// Brief: Master Arm Master Slave Control
FUNCTION_BLOCK PUBLIC FB_StateCtrlInit EXTENDS FB_MasterArmCtrlBase
VAR_INPUT
END_VAR
VAR_OUTPUT
END_VAR
VAR

END_VAR

// override this function in each exact controller
METHOD PROTECTED calcCmdJntPos : BOOL

VAR_IN_OUT CONSTANT
	i_slaveIdx :INT;
	i_shoulderPose :ST_Frame;
	i_masterArm :FB_MasterArm;
	i_slaveStatus :ST_SlaveStatus;
END_VAR

VAR
	centerVel:LREAL;
//	curJntPos:Vec7d;
END_VAR
IF m_isFinished THEN
	RETURN;
END_IF

IF m_timePeriod > 1 THEN
	m_isFinished :=true;
END_IF
END_METHOD

METHOD PUBLIC init : BOOL
VAR_IN_OUT CONSTANT
	i_masterArm	:FB_MasterArm;
END_VAR
VAR_IN_OUT 
	r_masterArmCtrlCmd :ST_ArmCtrlCmds;
END_VAR

VAR
	i:INT;
END_VAR
SUPER^.Init(i_masterArm,r_masterArmCtrlCmd);
m_jntEnableFlag :=g_zeroVec7i;
END_METHOD

END_FUNCTION_BLOCK

(* stored: Version 1.1.0.1, ProductVersion 3.1.4024.11
   POU FB_StateCtrlInit: Id {2f1b91d8-ebd5-4b63-92d8-450fe3a94973}, SpecialFunc None
   Method calcCmdJntPos: Id {b37c9272-afc7-4cb0-8e50-360f85145053}
   Method init: Id {0eca198b-2030-4cc0-a250-a6bdc9d0e230} *)
